TYPE ST_StepMode :
STRUCT
	bStepMode: BOOL;  //module in step mode
	bStep	 : BOOL;  //Step by step
END_STRUCT
END_TYPE

(* stored: Version 1.1.0.1, ProductVersion 3.1.4022.12
   DUT ST_StepMode: Id {83b103ab-746d-4908-b955-fe8df74bed43} *)
